FUNCTION_BLOCK FB_CalculateGermaniumThickness
VAR
END_VAR


METHOD PUBLIC Calculate
VAR_INPUT
    fDesiredTransmission : LREAL; // [1]
    fPhotonEnergy : LREAL; // [eV]
END_VAR
VAR_OUTPUT
    fThickness : LREAL; // [mm]
END_VAR
END_METHOD

END_FUNCTION_BLOCK

(* stored: Version 1.1.0.1
   POU FB_CalculateGermaniumThickness: Id {e3e3a7fb-d8d9-4b0b-a639-04b2da1ccafd}, SpecialFunc None
   Method Calculate: Id {c5739e06-e7c5-4e98-b50b-7bc8aa2c70f5} *)
